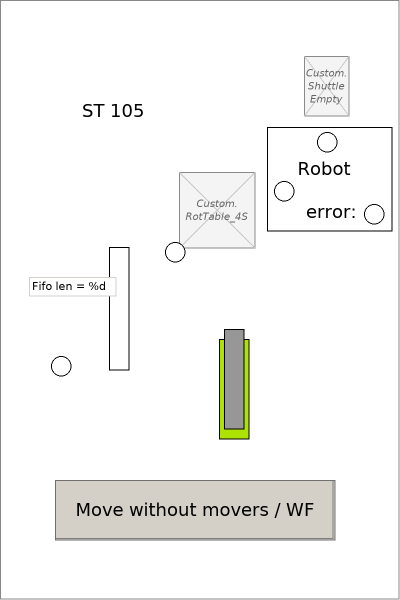
VISUALIZATION VISU_ST105  // 400x600
    Image (304,56 45x60), angle 90, invisible if: NOT __ISVALIDREF(GVL.st105_aut._Mover), image: Custom.Shuttle Empty
    Image (179,172 76x76), angle 45, image: Custom.RotTable_4S
        p2858320360: ST105_Axis.axis105_10W.rActPos
    Rectangle (109,247 20x123), angle 45
    Ellipse (51,356 20x20), colour toggle: GVL.st105_aut.fb_Feeder.simu_feeder.xOUT_NewPiece
    Ellipse (165,242 20x20), colour toggle: GVL.st105_aut.fb_Feeder.simu_feeder.xOUT_NewPiece
    Textfield (29,277 87x19), "Fifo len = %d", text variable: GVL.st105_aut.fb_Feeder.simu_fifo_feeder_to_rotTable.GetLen()
    Label (71,101 85x20), "ST 105"
    Rectangle (219,339 30x100)
    Rectangle (224,329 20x100)
        p2738717112: -GVL.st105_aut.fb_Pnp.fb_simu_axis105_11Z.rOUT_PixActual
    Button (55,480 280x60), "Move without movers / WF", colour toggle: HMI.bArForceCyclusState[StationList_e.ST105]
        tap HMI.btArForceCyclus[StationList_e.ST105].button
    Rectangle (267,127 125x104)
    Ellipse (274,181 20x20), colour toggle: GVL.st105_aut.fb_Pnp.aut_status_from_robot.Picked
    Ellipse (317,132 20x20), colour toggle: GVL.st105_aut.fb_Pnp.aut_status_from_robot.Placed
    Ellipse (364,204 20x20), colour toggle: GVL.st105_aut.fb_Pnp.fanuc_status.Fault
    Label (283,154 82x30), "Robot"
    Label (299,197 65x30), "error:"
END_VISUALIZATION

(* stored: Version 1.1.0.1, ProductVersion 3.1.4024.6
   Visu VISU_ST105: Id {b999b890-0911-46aa-a554-ca2d820bb3b0} *)
